(* CODESYS project Model.project

Project tree, tasks and I/O mapping:
  Device : CODESYS Control Win V3 x64, 3S - Smart Software Solutions GmbH, version 3.5.11.0
    application Application
      libraries: Standard, * (System); VisuDialogs, * (System); Util, * (System)
      task MainTask (cyclic, interval t#10ms, priority 1) calls Plant, Controller
      program Plant [ST]
      global variables GVL
      program Controller [ST]
      visualisation Visualization
      image pool ImagePool
  text list GlobalTextList
*)

// Device/Application/GVL
VAR_GLOBAL
	// Sensors:

	
	// Actuators:

END_VAR

// Device/Application/Plant
PROGRAM Plant

VAR CONSTANT
	// =========== Drum ===============
	DRUM_STEP : INT := 1;

	// =========== Heater ===============
	MAX_WATER_TEMPERATURE : INT := 100;
	MIN_WATER_TEMPERATURE : INT := 10;
	TEMPERATURE_STEP : INT := 1;
	
	// =========== Hatch lock device ===============
	HL_PIN_OFFSET : INT := 155;
	HL_PIN_STEP : INT := 5;
	
	// =========== Water control ===============
	FV_PIN_OFFSET : INT := 31;
	FV_PIN_STEP : INT := 5;
	WATER_STEP : REAL := 0.5;
	DRUM_HEIGHT : INT := 420;
END_VAR

VAR
	// =========== Drum ===============
	drum_angle : INT := 0; // The current rotation angle of the drum 

	// =========== Water control ===============
	rotor_state : BOOL := FALSE;		// Switch for rotor visualization
	fv_cur_offset : INT := 0; 			// Displacement of the filling valve pin
	water_level : REAL := 0;             // Current water level
	
	// =========== Hatch lock device ===============
	hl_cur_offset : INT := 0; 		   // Displacement of the pin of the hatch lock device
END_VAR

// ====================== DRUM ======================
// Operation of the tachometer
IF Controller.drum_state <> 0 THEN
	Controller.tachometer := TRUE;
ELSE
	Controller.tachometer := FALSE;
END_IF
	
// Emulation of the rotation of the drum
CASE Controller.drum_state OF
	1: drum_angle := (drum_angle + DRUM_STEP) MOD 360;
	2: drum_angle := (drum_angle - DRUM_STEP) MOD 360;
END_CASE
	
// ====================== HEATER ======================
// Emulation of heating and cooling of water
IF Controller.thermistor < MIN_WATER_TEMPERATURE THEN
	Controller.thermistor := MIN_WATER_TEMPERATURE;
END_IF

IF Controller.heater_on AND Controller.thermistor < MAX_WATER_TEMPERATURE THEN
	Controller.thermistor := Controller.thermistor + TEMPERATURE_STEP;	
ELSIF NOT Controller.heater_on AND Controller.thermistor > MIN_WATER_TEMPERATURE THEN
	Controller.thermistor := Controller.thermistor - 2 * TEMPERATURE_STEP;
END_IF
	
// ====================== HATCH LOCK DEVICE ======================
// Moving the pin
IF NOT Controller.hatch_lock_open AND hl_cur_offset > -HL_PIN_OFFSET THEN
	hl_cur_offset := hl_cur_offset - HL_PIN_STEP;
ELSIF Controller.hatch_lock_open AND hl_cur_offset < 0 THEN
	hl_cur_offset := hl_cur_offset + HL_PIN_STEP;
END_IF
	
// ====================== FILLING VALVE ======================	
IF Controller.filling_valve_open THEN 
		
	// Moving the pin to the open state
	IF fv_cur_offset < FV_PIN_OFFSET THEN
		fv_cur_offset := fv_cur_offset + FV_PIN_STEP;
	END_IF
		
	// Increasing the water level
	IF water_level < DRUM_HEIGHT THEN
		water_level := water_level + WATER_STEP;
	END_IF
	
// Moving the pin to the closed state 
ELSIF fv_cur_offset > 0 THEN
	fv_cur_offset := fv_cur_offset - FV_PIN_STEP;
END_IF	
	
// Operation of the pressostat
IF water_level >= DRUM_HEIGHT / 2 THEN
	Controller.pressostat := TRUE;
ELSE
	Controller.pressostat := FALSE;
END_IF
	
// ====================== DRAIN PUMP ======================	
IF Controller.drain_pump_on = TRUE THEN
		
	// Rotation of the rotor
	IF rotor_state = FALSE THEN
		rotor_state := TRUE;
	ELSE
		rotor_state := FALSE;
	END_IF
		
	// Decreasing the water level
	IF water_level > 0 THEN
		water_level := water_level - WATER_STEP;
	END_IF
		
END_IF

END_PROGRAM

// Device/Application/Controller
PROGRAM Controller

VAR_INPUT
	start_button : BOOL;
	temperature_button : BOOL;
	power_button : BOOL;
	hatch_lock_switch : BOOL;
	thermistor : INT;
	pressostat : BOOL;
	tachometer : BOOL;
END_VAR

VAR_OUTPUT
	temperature_led0 : BOOL;
	temperature_led1 : BOOL;
	temperature_led2 : BOOL;
	temperature_led3 : BOOL;
	washing_state_led0 : BOOL;
	washing_state_led1 : BOOL;
	washing_state_led2 : BOOL;
	washing_state_led3 : BOOL;
	washing_state_led4 : BOOL;
	error_led : BOOL;
	drum_state : INT;
	filling_valve_open : BOOL;
	hatch_lock_open : BOOL;
	drain_pump_on : BOOL;
	heater_on : BOOL;
END_VAR

VAR CONSTANT
	_P_INIT_S_BEGIN : INT := 0;
	_P_CONTROL_PANEL_S_INIT : INT := 0;
	_P_CONTROL_PANEL_S_WAIT : INT := 1;
	_P_CONTROL_PANEL_S_BUTTON_CONTROL : INT := 2;
	_P_CONTROL_PANEL_S_TEMPERATURE_CHANGE : INT := 3;
	_P_CONTROL_PANEL_S_HATCH_LOCK_CONTROL : INT := 4;
	_P_CONTROL_PANEL_S_START_WASHING : INT := 5;
	_P_INDICATION_S_WAIT : INT := 0;
	_P_INDICATION_S_INDICATE : INT := 1;
	_P_WASHING_PROCESS_S_WAIT : INT := 0;
	_P_WASHING_PROCESS_S_SUPPLY : INT := 1;
	_P_WASHING_PROCESS_S_WASHING : INT := 2;
	_P_WASHING_PROCESS_S_RELEASE : INT := 3;
	_P_WASHING_PROCESS_S_WATER_EXTRACTION : INT := 4;
	_P_WASHING_PROCESS_S_FINISHING : INT := 5;
	_P_TEMPERATURE_CONTROL_S_WAIT : INT := 0;
	_P_TEMPERATURE_CONTROL_S_WORK : INT := 1;
	_P_FILLING_VALVE_CONTROL_S_WORK : INT := 0;
	_P_ERROR_CONTROL_S_WAIT : INT := 0;
	_P_ERROR_CONTROL_S_ERROR : INT := 1;
	_P_HATCH_LOCK_CHECK_S_CHECK : INT := 0;
	_P_DRUM_CHECK_S_WAIT : INT := 0;
	_P_DRUM_CHECK_S_CHECK : INT := 1;
	_P_FILLING_VALVE_CHECK_S_WAIT : INT := 0;
	_P_FILLING_VALVE_CHECK_S_CHECK : INT := 1;
	_P_HEATER_CHECK_S_WAIT : INT := 0;
	_P_HEATER_CHECK_S_CHECK : INT := 1;
	_P_DRAIN_PUMP_CHECK_S_WAIT : INT := 0;
	_P_DRAIN_PUMP_CHECK_S_CHECK : INT := 1;
	_STOP : INT := 254;
	_ERROR : INT := 255;
END_VAR

VAR
	temperature : INT := 30;
	washing_started : BOOL;
	washing_state : INT := 0;
	error : BOOL;
	_p_Control_panel_v_prev_temp_btn_state : BOOL;
	_p_Control_panel_v_prev_start_btn_state : BOOL;
	_p_Washing_process_v_dir_changes_cnt : INT;
	_p_Error_control_v_prev_error : BOOL;
	_p_Filling_valve_check_v_prev_filling_valve : BOOL;
	_p_Heater_check_v_prev_heater : BOOL;
	_p_Heater_check_v_prev_temperature : INT;
	_p_Drain_pump_check_v_prev_drain_pump : BOOL;
	_global_time : TIME;
	_g_p_Washing_process_time : TIME;
	_g_p_Drum_check_time : TIME;
	_g_p_Filling_valve_check_time : TIME;
	_g_p_Heater_check_time : TIME;
	_g_p_Drain_pump_check_time : TIME;
	_g_p_Init_state : INT := _P_INIT_S_BEGIN;
	_g_p_Control_panel_state : INT := _STOP;
	_g_p_Indication_state : INT := _STOP;
	_g_p_Washing_process_state : INT := _STOP;
	_g_p_Temperature_control_state : INT := _STOP;
	_g_p_Filling_valve_control_state : INT := _STOP;
	_g_p_Error_control_state : INT := _STOP;
	_g_p_Hatch_lock_check_state : INT := _STOP;
	_g_p_Drum_check_state : INT := _STOP;
	_g_p_Filling_valve_check_state : INT := _STOP;
	_g_p_Heater_check_state : INT := _STOP;
	_g_p_Drain_pump_check_state : INT := _STOP;
END_VAR

_global_time := TIME();

CASE _g_p_Init_state OF
	_P_INIT_S_BEGIN:
		_g_p_Control_panel_state := _P_CONTROL_PANEL_S_INIT;
		_g_p_Indication_state := _P_INDICATION_S_WAIT;
		_g_p_Washing_process_state := _P_WASHING_PROCESS_S_WAIT;
		_g_p_Temperature_control_state := _P_TEMPERATURE_CONTROL_S_WAIT;
		_g_p_Filling_valve_control_state := _P_FILLING_VALVE_CONTROL_S_WORK;
		_g_p_Error_control_state := _P_ERROR_CONTROL_S_WAIT;
		_g_p_Drum_check_state := _P_DRUM_CHECK_S_WAIT;
		_g_p_Heater_check_state := _P_HEATER_CHECK_S_WAIT;
		_g_p_Drain_pump_check_state := _P_DRAIN_PUMP_CHECK_S_WAIT;
		_g_p_Hatch_lock_check_state := _P_HATCH_LOCK_CHECK_S_CHECK;
		_g_p_Filling_valve_check_state := _P_FILLING_VALVE_CHECK_S_WAIT;
		_g_p_Init_state := _STOP;
END_CASE

CASE _g_p_Control_panel_state OF
	_P_CONTROL_PANEL_S_INIT:
		_p_Control_panel_v_prev_temp_btn_state := temperature_button;
		_p_Control_panel_v_prev_start_btn_state := start_button;
		hatch_lock_open := TRUE;
		_g_p_Control_panel_state := _P_CONTROL_PANEL_S_WAIT;
	_P_CONTROL_PANEL_S_WAIT:
		IF NOT power_button THEN
			washing_state := 0;
			temperature := 30;
			drum_state := 0;
			filling_valve_open := FALSE;
			washing_started := FALSE;
			hatch_lock_open := TRUE;
			drain_pump_on := FALSE;
			heater_on := FALSE;
			error := FALSE;
		ELSIF NOT washing_started THEN
			_g_p_Control_panel_state := _P_CONTROL_PANEL_S_BUTTON_CONTROL;
		END_IF
	_P_CONTROL_PANEL_S_BUTTON_CONTROL:
		IF temperature_button AND NOT _p_Control_panel_v_prev_temp_btn_state THEN
			_g_p_Control_panel_state := _P_CONTROL_PANEL_S_TEMPERATURE_CHANGE;
		ELSIF start_button AND NOT _p_Control_panel_v_prev_start_btn_state THEN
			_g_p_Control_panel_state := _P_CONTROL_PANEL_S_HATCH_LOCK_CONTROL;
		ELSE
			_g_p_Control_panel_state := _P_CONTROL_PANEL_S_WAIT;
		END_IF
		_p_Control_panel_v_prev_start_btn_state := start_button;
		_p_Control_panel_v_prev_temp_btn_state := temperature_button;
	_P_CONTROL_PANEL_S_TEMPERATURE_CHANGE:
		CASE temperature OF
			30:
				temperature := 40;
			40:
				temperature := 60;
			60:
				temperature := 95;
			95:
				temperature := 30;
		END_CASE
		_g_p_Control_panel_state := _P_CONTROL_PANEL_S_WAIT;
	_P_CONTROL_PANEL_S_HATCH_LOCK_CONTROL:
		IF hatch_lock_switch THEN
			hatch_lock_open := FALSE;
			error := FALSE;
			_g_p_Control_panel_state := _P_CONTROL_PANEL_S_START_WASHING;
		ELSE
			error := TRUE;
			_g_p_Control_panel_state := _P_CONTROL_PANEL_S_WAIT;
		END_IF
	_P_CONTROL_PANEL_S_START_WASHING:
		washing_started := TRUE;
		filling_valve_open := TRUE;
		washing_state := 1;
		_g_p_Control_panel_state := _P_CONTROL_PANEL_S_WAIT;
END_CASE

CASE _g_p_Indication_state OF
	_P_INDICATION_S_WAIT:
		IF NOT power_button THEN
			temperature_led0 := FALSE;
			temperature_led1 := FALSE;
			temperature_led2 := FALSE;
			temperature_led3 := FALSE;
			washing_state_led0 := FALSE;
			washing_state_led1 := FALSE;
			washing_state_led2 := FALSE;
			washing_state_led3 := FALSE;
			washing_state_led4 := FALSE;
			error_led := FALSE;
		ELSE
			_g_p_Indication_state := _P_INDICATION_S_INDICATE;
		END_IF
	_P_INDICATION_S_INDICATE:
		CASE temperature OF
			30:
				temperature_led0 := TRUE;
				temperature_led1 := FALSE;
				temperature_led2 := FALSE;
				temperature_led3 := FALSE;
			40:
				temperature_led0 := FALSE;
				temperature_led1 := TRUE;
				temperature_led2 := FALSE;
				temperature_led3 := FALSE;
			60:
				temperature_led0 := FALSE;
				temperature_led1 := FALSE;
				temperature_led2 := TRUE;
				temperature_led3 := FALSE;
			95:
				temperature_led0 := FALSE;
				temperature_led1 := FALSE;
				temperature_led2 := FALSE;
				temperature_led3 := TRUE;
		END_CASE
		CASE washing_state OF
			0:
				washing_state_led0 := FALSE;
				washing_state_led1 := FALSE;
				washing_state_led2 := FALSE;
				washing_state_led3 := FALSE;
				washing_state_led4 := FALSE;
			1:
				washing_state_led0 := TRUE;
				washing_state_led1 := FALSE;
				washing_state_led2 := FALSE;
				washing_state_led3 := FALSE;
				washing_state_led4 := FALSE;
			2:
				washing_state_led0 := FALSE;
				washing_state_led1 := TRUE;
				washing_state_led2 := FALSE;
				washing_state_led3 := FALSE;
				washing_state_led4 := FALSE;
			3:
				washing_state_led0 := FALSE;
				washing_state_led1 := FALSE;
				washing_state_led2 := TRUE;
				washing_state_led3 := FALSE;
				washing_state_led4 := FALSE;
			4:
				washing_state_led0 := FALSE;
				washing_state_led1 := FALSE;
				washing_state_led2 := FALSE;
				washing_state_led3 := TRUE;
				washing_state_led4 := FALSE;
			5:
				washing_state_led0 := FALSE;
				washing_state_led1 := FALSE;
				washing_state_led2 := FALSE;
				washing_state_led3 := FALSE;
				washing_state_led4 := TRUE;
		END_CASE
		IF error THEN
			error_led := TRUE;
		ELSE
			error_led := FALSE;
		END_IF
		_g_p_Indication_state := _P_INDICATION_S_WAIT;
END_CASE

CASE _g_p_Washing_process_state OF
	_P_WASHING_PROCESS_S_WAIT:
		CASE washing_state OF
			1:
				_g_p_Washing_process_state := _P_WASHING_PROCESS_S_SUPPLY;
			2:
				_g_p_Washing_process_time := _global_time;
				_g_p_Washing_process_state := _P_WASHING_PROCESS_S_WASHING;
			3:
				_g_p_Washing_process_time := _global_time;
				_g_p_Washing_process_state := _P_WASHING_PROCESS_S_RELEASE;
			4:
				_g_p_Washing_process_time := _global_time;
				_g_p_Washing_process_state := _P_WASHING_PROCESS_S_WATER_EXTRACTION;
			5:
				_g_p_Washing_process_time := _global_time;
				_g_p_Washing_process_state := _P_WASHING_PROCESS_S_FINISHING;
		END_CASE
	_P_WASHING_PROCESS_S_SUPPLY:
		IF pressostat AND thermistor > temperature - 2 THEN
			washing_state := 2;
			drum_state := 1;
		END_IF
		_g_p_Washing_process_state := _P_WASHING_PROCESS_S_WAIT;
	_P_WASHING_PROCESS_S_WASHING:
		IF NOT power_button OR error THEN
			_g_p_Washing_process_time := _global_time;
			_g_p_Washing_process_state := _P_WASHING_PROCESS_S_WAIT;
		END_IF
		IF (_global_time - _g_p_Washing_process_time) >= T#7s THEN
			IF drum_state = 2 THEN
				drum_state := 1;
				washing_state := 3;
				drain_pump_on := TRUE;
				_g_p_Washing_process_state := _P_WASHING_PROCESS_S_WAIT;
			ELSE
				drum_state := 2;
				_g_p_Washing_process_time := _global_time;
			END_IF
		END_IF
	_P_WASHING_PROCESS_S_RELEASE:
		IF NOT power_button OR error THEN
			_g_p_Washing_process_time := _global_time;
			_g_p_Washing_process_state := _P_WASHING_PROCESS_S_WAIT;
		END_IF
		IF (_global_time - _g_p_Washing_process_time) >= T#15s THEN
			washing_state := 4;
			_g_p_Washing_process_state := _P_WASHING_PROCESS_S_WAIT;
		END_IF
	_P_WASHING_PROCESS_S_WATER_EXTRACTION:
		IF _p_Washing_process_v_dir_changes_cnt = 4 THEN
			washing_state := 5;
			drum_state := 0;
			drain_pump_on := FALSE;
			_g_p_Washing_process_state := _P_WASHING_PROCESS_S_WAIT;
		END_IF
		IF NOT power_button OR error THEN
			_p_Washing_process_v_dir_changes_cnt := 0;
			_g_p_Washing_process_time := _global_time;
			_g_p_Washing_process_state := _P_WASHING_PROCESS_S_WAIT;
		END_IF
		IF (_global_time - _g_p_Washing_process_time) >= T#5s THEN
			_p_Washing_process_v_dir_changes_cnt := _p_Washing_process_v_dir_changes_cnt + 1;
			IF drum_state = 1 THEN
				drum_state := 2;
			ELSE
				drum_state := 1;
			END_IF
			_g_p_Washing_process_time := _global_time;
		END_IF
	_P_WASHING_PROCESS_S_FINISHING:
		IF (_global_time - _g_p_Washing_process_time) >= T#2s THEN
			hatch_lock_open := TRUE;
			washing_started := FALSE;
			washing_state := 0;
			_g_p_Washing_process_state := _P_WASHING_PROCESS_S_WAIT;
		END_IF
END_CASE

CASE _g_p_Temperature_control_state OF
	_P_TEMPERATURE_CONTROL_S_WAIT:
		IF washing_state = 1 OR washing_state = 2 THEN
			_g_p_Temperature_control_state := _P_TEMPERATURE_CONTROL_S_WORK;
		ELSE
			heater_on := FALSE;
		END_IF
	_P_TEMPERATURE_CONTROL_S_WORK:
		IF thermistor < temperature THEN
			heater_on := TRUE;
		ELSE
			heater_on := FALSE;
		END_IF
		_g_p_Temperature_control_state := _P_TEMPERATURE_CONTROL_S_WAIT;
END_CASE

CASE _g_p_Filling_valve_control_state OF
	_P_FILLING_VALVE_CONTROL_S_WORK:
		IF pressostat THEN
			filling_valve_open := FALSE;
		END_IF
END_CASE

CASE _g_p_Error_control_state OF
	_P_ERROR_CONTROL_S_WAIT:
		IF error AND NOT _p_Error_control_v_prev_error THEN
			_g_p_Error_control_state := _P_ERROR_CONTROL_S_ERROR;
		END_IF
		_p_Error_control_v_prev_error := error;
	_P_ERROR_CONTROL_S_ERROR:
		drum_state := 0;
		washing_state := 0;
		filling_valve_open := FALSE;
		washing_started := FALSE;
		drain_pump_on := FALSE;
		heater_on := FALSE;
		_g_p_Error_control_state := _P_ERROR_CONTROL_S_WAIT;
END_CASE

CASE _g_p_Hatch_lock_check_state OF
	_P_HATCH_LOCK_CHECK_S_CHECK:
		IF NOT hatch_lock_switch AND washing_state > 0 THEN
			error := TRUE;
		END_IF
END_CASE

CASE _g_p_Drum_check_state OF
	_P_DRUM_CHECK_S_WAIT:
		IF drum_state <> 0 THEN
			_g_p_Drum_check_time := _global_time;
			_g_p_Drum_check_state := _P_DRUM_CHECK_S_CHECK;
		END_IF
	_P_DRUM_CHECK_S_CHECK:
		IF tachometer THEN
			_g_p_Drum_check_state := _P_DRUM_CHECK_S_WAIT;
		END_IF
		IF (_global_time - _g_p_Drum_check_time) >= T#1s THEN
			error := TRUE;
			_g_p_Drum_check_state := _P_DRUM_CHECK_S_WAIT;
		END_IF
END_CASE

CASE _g_p_Filling_valve_check_state OF
	_P_FILLING_VALVE_CHECK_S_WAIT:
		IF filling_valve_open AND NOT _p_Filling_valve_check_v_prev_filling_valve THEN
			_g_p_Filling_valve_check_time := _global_time;
			_g_p_Filling_valve_check_state := _P_FILLING_VALVE_CHECK_S_CHECK;
		END_IF
		_p_Filling_valve_check_v_prev_filling_valve := filling_valve_open;
	_P_FILLING_VALVE_CHECK_S_CHECK:
		IF pressostat OR NOT filling_valve_open THEN
			_g_p_Filling_valve_check_state := _P_FILLING_VALVE_CHECK_S_WAIT;
		END_IF
		IF (_global_time - _g_p_Filling_valve_check_time) >= T#5s THEN
			error := TRUE;
			_g_p_Filling_valve_check_state := _P_FILLING_VALVE_CHECK_S_WAIT;
		END_IF
END_CASE

CASE _g_p_Heater_check_state OF
	_P_HEATER_CHECK_S_WAIT:
		IF heater_on AND NOT _p_Heater_check_v_prev_heater THEN
			_g_p_Heater_check_time := _global_time;
			_g_p_Heater_check_state := _P_HEATER_CHECK_S_CHECK;
		END_IF
		_p_Heater_check_v_prev_heater := heater_on;
	_P_HEATER_CHECK_S_CHECK:
		IF NOT heater_on THEN
			_g_p_Heater_check_state := _P_HEATER_CHECK_S_WAIT;
		END_IF
		IF (_global_time - _g_p_Heater_check_time) >= T#1s THEN
			IF thermistor - _p_Heater_check_v_prev_temperature <= 0 THEN
				error := TRUE;
			END_IF
			_g_p_Heater_check_state := _P_HEATER_CHECK_S_WAIT;
		END_IF
END_CASE

CASE _g_p_Drain_pump_check_state OF
	_P_DRAIN_PUMP_CHECK_S_WAIT:
		IF drain_pump_on AND NOT _p_Drain_pump_check_v_prev_drain_pump THEN
			_g_p_Drain_pump_check_time := _global_time;
			_g_p_Drain_pump_check_state := _P_DRAIN_PUMP_CHECK_S_CHECK;
		END_IF
		_p_Drain_pump_check_v_prev_drain_pump := drain_pump_on;
	_P_DRAIN_PUMP_CHECK_S_CHECK:
		IF NOT drain_pump_on THEN
			_g_p_Drain_pump_check_state := _P_DRAIN_PUMP_CHECK_S_WAIT;
		END_IF
		IF (_global_time - _g_p_Drain_pump_check_time) >= T#5s THEN
			IF pressostat THEN
				error := TRUE;
			END_IF
			_g_p_Drain_pump_check_state := _P_DRAIN_PUMP_CHECK_S_WAIT;
		END_IF
END_CASE

END_PROGRAM

// Device/Application/Visualization
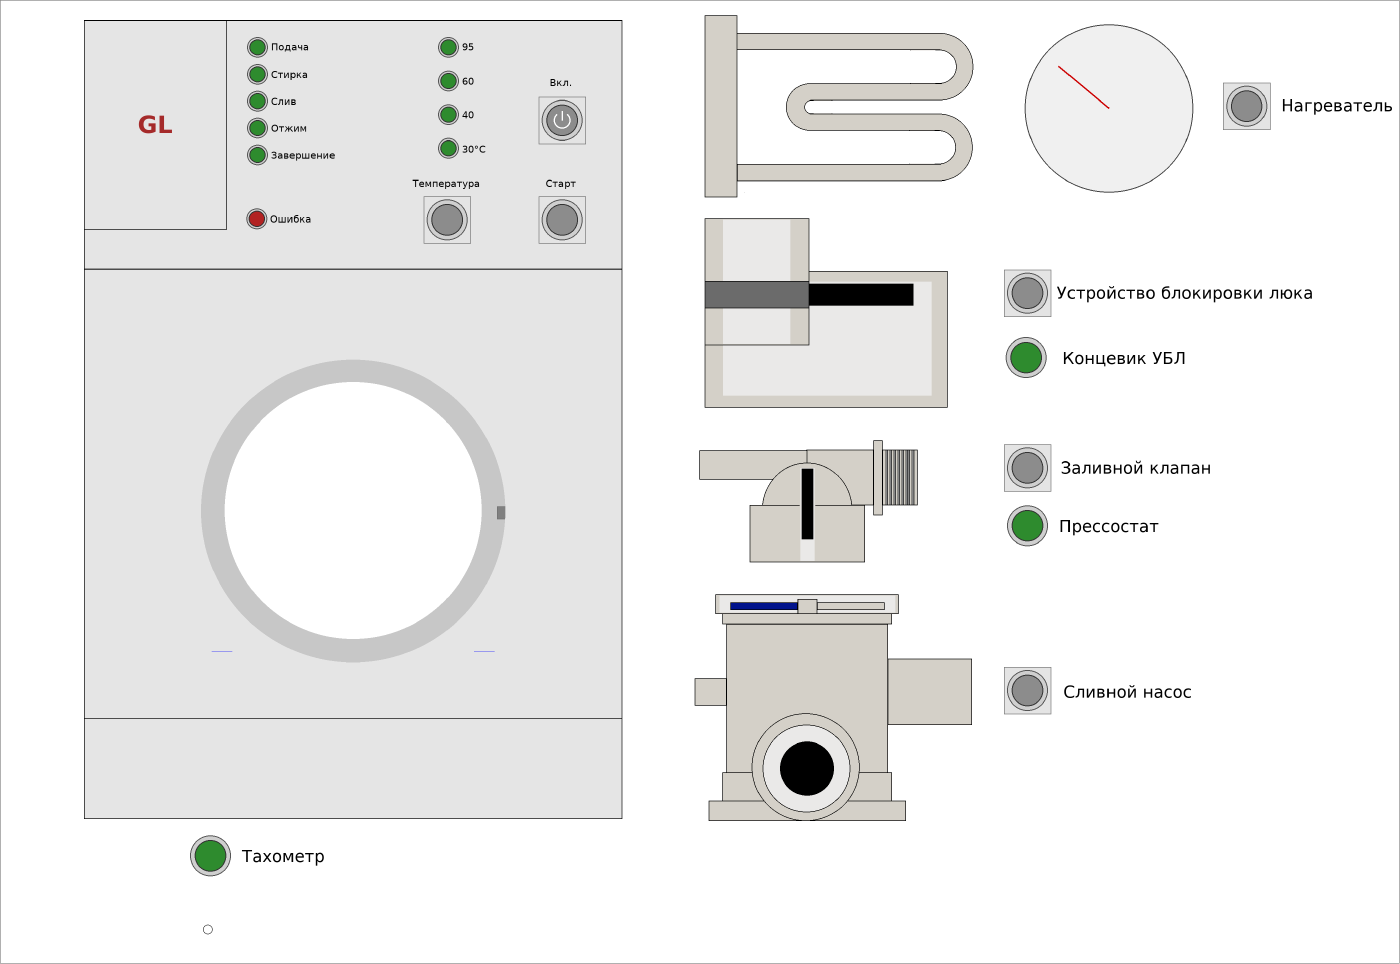
VISUALIZATION Visualization  // 2082x1434
    Rectangle (125,400 800x800)
    Rectangle (125,30 800x370)
    PowerSwitch (801,144 70x70), variable: Controller.power_button, behaviour: TOGGLE, style: Switch-PowerSwitch-Gray
    PushSwitch (630,292 70x70), variable: Controller.temperature_button, behaviour: TAP, style: Switch-PushSwitch-Gray
    Lamp1 (645,53 44x35), variable: Controller.temperature_led3, style: Lamp-Lamp1-Green
    Lamp1 (645,103 44x35), variable: Controller.temperature_led2, style: Lamp-Lamp1-Green
    Lamp1 (645,153 44x35), variable: Controller.temperature_led1, style: Lamp-Lamp1-Green
    Lamp1 (645,203 44x35), variable: Controller.temperature_led0, style: Lamp-Lamp1-Green
    Label (759,108 150x30), "Вкл."
    Label (589,258 150x30), "Температура"
    PushSwitch (801,292 70x70), variable: Controller.start_button, behaviour: TAP, style: Switch-PushSwitch-Gray
    Label (759,258 150x30), "Старт"
    Label (678,55 36x30), "95"
    Label (678,106 36x30), "60"
    Label (678,156 36x30), "40"
    Label (672,207 66x30), "30°C"
    Lamp1 (361,53 44x35), variable: Controller.washing_state_led0, style: Lamp-Lamp1-Green
    Lamp1 (361,93 44x35), variable: Controller.washing_state_led1, style: Lamp-Lamp1-Green
    Lamp1 (361,133 44x35), variable: Controller.washing_state_led2, style: Lamp-Lamp1-Green
    Lamp1 (361,173 44x35), variable: Controller.washing_state_led3, style: Lamp-Lamp1-Green
    Label (400,55 74x30), "Подача"
    Label (400,96 67x30), "Стирка"
    Label (400,136 73x30), "Слив"
    Label (400,176 73x30), "Отжим"
    Lamp1 (361,213 44x35), variable: Controller.washing_state_led4, style: Lamp-Lamp1-Green
    Label (400,216 122x30), "Завершение"
    Lamp1 (360,308 44x35), variable: Controller.error_led, style: Lamp-Lamp1-Red
    Label (399,311 67x30), "Ошибка"
    Rectangle (125,1068 800x150)
    Rectangle (125,30 212x311), "GL"
    Ellipse (275,510 500x500)
    Ellipse (315,550 420x420)
        p2858320360: Plant.drum_angle
    Lamp1 (1010,286 194x0), style: Lamp-Lamp1-Yellow
    RadioButton (300,1333 456x99), variable: Controller.drum_state
        Areas[0]: Text=Drum_off
        Areas[1]: Text=Drum_clockwise
        Areas[2]: Text=Drum_counterclockwise
    Ellipse (1347,49 100x100), colour toggle: Controller.heater_on
    Ellipse (1372,74 50x50), colour toggle: Controller.heater_on
    Rectangle (1093,49 305x25), colour toggle: Controller.heater_on
    Ellipse (1373,75 48x48)
    Rectangle (1203,75 195x48)
    Rectangle (1396,50 4x23), colour toggle: Controller.heater_on
    Ellipse (1169,124 70x70), colour toggle: Controller.heater_on
    Rectangle (1205,124 195x25), colour toggle: Controller.heater_on
    Rectangle (1397,125 4x23), colour toggle: Controller.heater_on
    Ellipse (1346,169 100x100), colour toggle: Controller.heater_on
    Ellipse (1371,194 50x50), colour toggle: Controller.heater_on
    Rectangle (1204,169 193x25), colour toggle: Controller.heater_on
    Ellipse (1372,195 48x48)
    Rectangle (1202,195 195x48)
    Rectangle (1395,170 4x23), colour toggle: Controller.heater_on
    Rectangle (1096,244 303x25), colour toggle: Controller.heater_on
    Rectangle (1396,245 4x23), colour toggle: Controller.heater_on
    Ellipse (1196,149 20x20), colour toggle: Controller.heater_on
    Ellipse (1197,150 18x18)
    Rectangle (1205,150 195x18)
    Rectangle (1202,125 4x23), colour toggle: Controller.heater_on
    Rectangle (1202,170 4x23), colour toggle: Controller.heater_on
    RoundedRectangle (1048,23 48x270)
    PushSwitch (1819,123 70x70), variable: Controller.heater_on, behaviour: TOGGLE, style: Switch-PushSwitch-Gray
    Label (1897,145 183x24), "Нагреватель"
    PushSwitch (1493,661 70x70), variable: Controller.filling_valve_open, behaviour: TOGGLE, style: Switch-PushSwitch-Gray
    PushSwitch (1493,992 70x70), variable: Controller.drain_pump_on, behaviour: TOGGLE, style: Switch-PushSwitch-Gray
    Label (1569,684 241x24), "Заливной клапан"
    Label (1569,1015 216x29), "Сливной насос"
    RoundedRectangle (1048,403 361x203)
    PushSwitch (1493,401 70x70), variable: Controller.hatch_lock_open, behaviour: TOGGLE, style: Switch-PushSwitch-Gray
    Label (1569,418 387x36), "Устройство блокировки люка"
    RoundedRectangle (1074,418 312x171)
    RoundedRectangle (1031,342 188x155), angle 270
    Rectangle (1074,326 102x186)
    Meter360 (1524,36 250x250), value: Controller.thermistor, style: Meter-Meter360-Gray, scale format: %.1f, scale 0..100
        p518627256: ℃
    RoundedRectangle (1105,361 40x155), angle 270
    RoundedRectangle (1203,422 155x32)
        p3560616238: Plant.hl_cur_offset
    Rectangle (1199,669 100x82)
    Rectangle (1040,670 160x43), angle 180
    Ellipse (1133,688 134x141)
    RoundedRectangle (1115,751 171x85)
    RoundedRectangle (1074,911 252x17)
    Rectangle (1089,919 222x240), angle 270
    Rectangle (1333,967 98x125), angle 270
    Rectangle (1036,1006 40x47), angle 270
    RoundedRectangle (1074,1149 252x46)
    RoundedRectangle (1054,1191 293x30)
    RoundedRectangle (1064,884 272x29)
    Ellipse (1118,1061 160x160)
    Ellipse (1134,1078 130x130)
    Ellipse (1160,1103 80x80)
    RoundedRectangle (1069,885 263x27)
    RoundedRectangle (1186,891 29x22)
    Rectangle (1260,852 11x100), angle 270, colour toggle: Plant.rotor_state
    Rectangle (1131,852 11x100), angle 270, colour toggle: Plant.rotor_state
    Rectangle (1299,655 13x111)
    Rectangle (1312,669 52x82)
    Rectangle (1329,669 3x82)
    Rectangle (1335,669 3x82)
    Rectangle (1341,669 3x82)
    Rectangle (1347,669 3x82)
    Rectangle (1350,669 3x82)
    Rectangle (1356,669 3x82)
    Rectangle (1317,669 3x82)
    Rectangle (1323,669 3x82)
    Rectangle (1189,695 23x140)
    RoundedRectangle (1149,741 105x17), angle 90
        p2738717112: Plant.fv_cur_offset
    Rectangle (315,969 420x0)
        p2773130477: -Plant.water_level
    Lamp1 (1491,497 70x70), variable: Controller.hatch_lock_switch, style: Lamp-Lamp1-Green
    Label (1577,515 233x36), "Концевик УБЛ"
    Lamp1 (1493,747 70x70), variable: Controller.pressostat, style: Lamp-Lamp1-Green
    Label (1572,765 158x36), "Прессостат"
    Lamp1 (278,1238 70x70), variable: Controller.tachometer, style: Lamp-Lamp1-Green
    Label (357,1256 158x36), "Тахометр"
    Ellipse (294,528 462x462)
    Button (739,753 34x19)
        toggle Controller.hatch_lock_switch
    Ellipse (249,485 552x550)
END_VISUALIZATION
